(* Logix 5000 project; controller ICA02 vendor 1 type 14 code 150 rev 37.11; software revision 37.00 *)

TASK MainTask (continuous, watchdog 500 ms) : MainProgram

MODULES
   Local : vendor 1 type 14 code 150 (Compact 0, rev 37.11)
      Discrete_IO : Embedded (Compact 1, rev 3.1, Output RPI 20 ms)
      Analog_IO : Embedded (Compact 2, rev 1.1, Output RPI 80 ms)
      Counters : Embedded (Compact 3, rev 1.1, Output RPI 20 ms)
END_MODULES

VAR_GLOBAL   (* controller tags *)
   LSL : ALIAS FOR Local:1:I.Data.12;
   M1 : ALIAS FOR Local:1:O.Data.1;
   M2 : ALIAS FOR Local:1:O.Data.0;
   M3 : ALIAS FOR Local:1:O.Data.2;
   Start : ALIAS FOR Local:1:I.Data.11;
   Stop : ALIAS FOR Local:1:I.Data.8;
END_VAR

PROGRAM MainProgram   (* main routine MainRoutine *)

ROUTINE MainRoutine   (* ladder *)
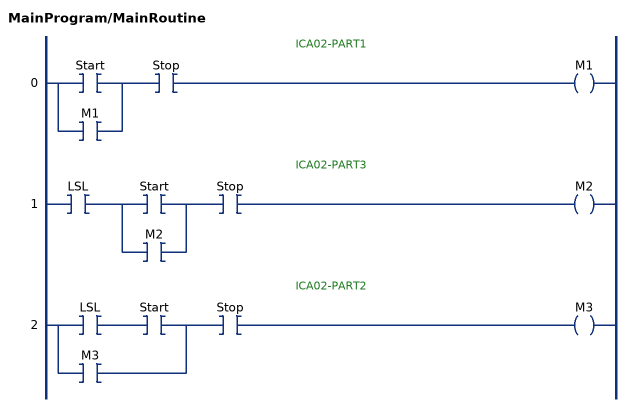
   // ICA02-PART1
   0: [XIC(Start) ,XIC(M1) ]XIC(Stop)OTE(M1);
   // ICA02-PART3
   1: XIC(LSL)[XIC(Start) ,XIC(M2) ]XIC(Stop)OTE(M2);
   // ICA02-PART2
   2: [XIC(LSL) XIC(Start) ,XIC(M3) ]XIC(Stop)OTE(M3);
END_ROUTINE
END_PROGRAM
